FUNCTION_BLOCK FB_Coordinador_SFC EXTENDS FB_Object_Template_SFC;
VAR_INPUT
 
//Discharger
	Discharger_Ready: BOOL;
	Discharger_Done: BOOL;

	
//Elevador
	Elevator_B1_Ready:BOOL;
	Elevator_B2_Ready:BOOL;
	Elevator_S_Ready:BOOL;
	
	Elevator_B1_Done:BOOL;
	Elevator_B2_Done:BOOL;
	Elevator_S_Done:BOOL;

//Conveyors
	Conveyor_B1_Ready:BOOL;
	Conveyor_B2_Ready:BOOL;
	Conveyor_S_Ready:BOOL;
	
	Conveyor_B1_Done:BOOL;
	Conveyor_B2_Done:BOOL;
	Conveyor_S_Done:BOOL;
	
	Elevator_B1_END_Down:BOOL;
	Elevator_B2_END_Down:BOOL;
	Elevator_S_END_Down:BOOL;
	
	B1 :BOOL;

END_VAR
VAR_OUTPUT
	//Discharger
	Discharger_Ack: BOOL;
	Discharger_Execute: BOOL;
	
	//Elevador
	Elevator_B1_Execute:BOOL;
	Elevator_B2_Execute:BOOL;
	Elevator_S_Execute:BOOL;
	
	Elevator_B1_Up:BOOL;
	Elevator_B2_Up:BOOL;
	Elevator_S_Up:BOOL;
	
	Elevator_B1_Down:BOOL;
	Elevator_B2_Down:BOOL;
	Elevator_S_Down:BOOL;
	Elevator_S_Step:BOOL;
	
	Elevator_B1_Ack:BOOL;
	Elevator_B2_Ack:BOOL;
	Elevator_S_Ack:BOOL;

//Conveyor
	Conveyor_B1_Execute:BOOL;
	Conveyor_B2_Execute:BOOL;
	Conveyor_S_Execute:BOOL;
	
	Conveyor_B1_Ack:BOOL;
	Conveyor_B2_Ack:BOOL;
	Conveyor_S_Ack:BOOL;
	
	Conveyor_B1_Proces:BOOL;
	Conveyor_B2_Proces:BOOL;
	Conveyor_S_Dischar:BOOL;
	
END_VAR
VAR

//Cuenta de bandejas
	Count:INT;

END_VAR

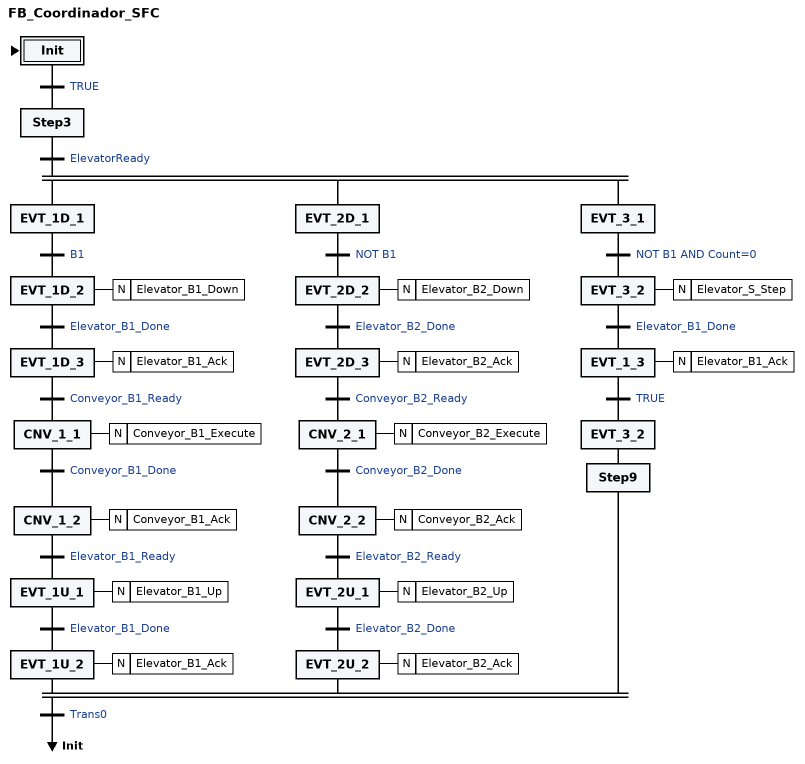
INITIAL_STEP Init:
END_STEP
TRANSITION FROM Init TO Step3
    := TRUE;
END_TRANSITION
STEP Step3:
END_STEP
TRANSITION FROM Step3 TO (EVT_1D_1, EVT_2D_1, EVT_3_1)
    := ElevatorReady;
END_TRANSITION
STEP EVT_1D_1:
END_STEP
TRANSITION FROM EVT_1D_1 TO EVT_1D_2
    := B1;
END_TRANSITION
STEP EVT_1D_2:
    Elevator_B1_Down(N);
END_STEP
TRANSITION FROM EVT_1D_2 TO EVT_1D_3
    := Elevator_B1_Done;
END_TRANSITION
STEP EVT_1D_3:
    Elevator_B1_Ack(N);
END_STEP
TRANSITION FROM EVT_1D_3 TO CNV_1_1
    := Conveyor_B1_Ready;
END_TRANSITION
STEP CNV_1_1:
    Conveyor_B1_Execute(N);
END_STEP
TRANSITION FROM CNV_1_1 TO CNV_1_2
    := Conveyor_B1_Done;
END_TRANSITION
STEP CNV_1_2:
    Conveyor_B1_Ack(N);
END_STEP
TRANSITION FROM CNV_1_2 TO EVT_1U_1
    := Elevator_B1_Ready;
END_TRANSITION
STEP EVT_1U_1:
    Elevator_B1_Up(N);
END_STEP
TRANSITION FROM EVT_1U_1 TO EVT_1U_2
    := Elevator_B1_Done;
END_TRANSITION
STEP EVT_1U_2:
    Elevator_B1_Ack(N);
END_STEP
STEP EVT_2D_1:
END_STEP
TRANSITION FROM EVT_2D_1 TO EVT_2D_2
    := NOT B1;
END_TRANSITION
STEP EVT_2D_2:
    Elevator_B2_Down(N);
END_STEP
TRANSITION FROM EVT_2D_2 TO EVT_2D_3
    := Elevator_B2_Done;
END_TRANSITION
STEP EVT_2D_3:
    Elevator_B2_Ack(N);
END_STEP
TRANSITION FROM EVT_2D_3 TO CNV_2_1
    := Conveyor_B2_Ready;
END_TRANSITION
STEP CNV_2_1:
    Conveyor_B2_Execute(N);
END_STEP
TRANSITION FROM CNV_2_1 TO CNV_2_2
    := Conveyor_B2_Done;
END_TRANSITION
STEP CNV_2_2:
    Conveyor_B2_Ack(N);
END_STEP
TRANSITION FROM CNV_2_2 TO EVT_2U_1
    := Elevator_B2_Ready;
END_TRANSITION
STEP EVT_2U_1:
    Elevator_B2_Up(N);
END_STEP
TRANSITION FROM EVT_2U_1 TO EVT_2U_2
    := Elevator_B2_Done;
END_TRANSITION
STEP EVT_2U_2:
    Elevator_B2_Ack(N);
END_STEP
STEP EVT_3_1:
END_STEP
TRANSITION FROM EVT_3_1 TO EVT_3_2
    := NOT B1 AND Count=0;
END_TRANSITION
STEP EVT_3_2:
    Elevator_S_Step(N);
END_STEP
TRANSITION FROM EVT_3_2 TO EVT_1_3
    := Elevator_B1_Done;
END_TRANSITION
STEP EVT_1_3:
    Elevator_B1_Ack(N);
END_STEP
TRANSITION FROM EVT_1_3 TO EVT_3_2
    := TRUE;
END_TRANSITION
STEP EVT_3_2:
END_STEP
// no transition between EVT_3_2 and Step9
STEP Step9:
END_STEP
TRANSITION FROM (EVT_1U_2, EVT_2U_2, Step9) TO Init
    := Trans0;
END_TRANSITION

TRANSITION ElevatorReady:
Elevator_B1_Ready OR Elevator_B2_Ready OR Elevator_S_Ready;
END_TRANSITION

END_FUNCTION_BLOCK

(* stored: Version 1.1.0.1, ProductVersion 3.1.4024.6
   POU FB_Coordinador_SFC: Id {d10e6de2-55ea-46a1-9897-87bb74187acf}, SpecialFunc None
   Transition ElevatorReady: Id {a9ca3384-6594-4c89-bfb7-0676ac08e5ee} *)
